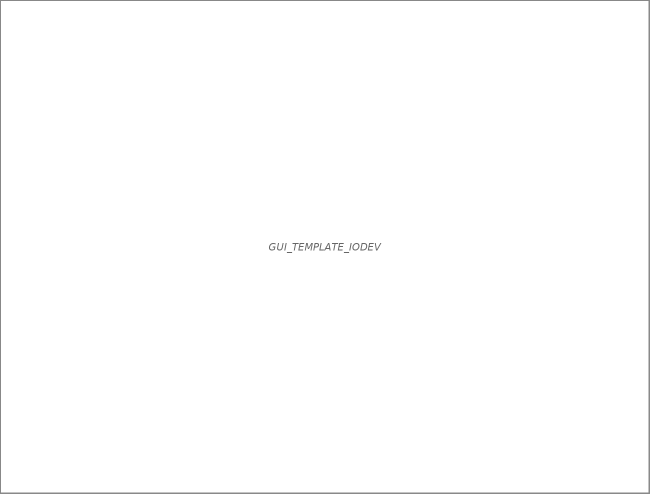
VISUALIZATION GUI_IODev002  // 650x494
    Frame (0,0 650x494)
        shows GUI_TEMPLATE_IODEV(m_Instance := MAIN.IODev002)
END_VISUALIZATION

(* stored: Version 1.1.0.1, ProductVersion 3.1.4024.3
   Visu GUI_IODev002: Id {e523f841-3b7e-491b-b311-44f46bfd5b7c} *)
